// TIA Portal V15.1 export
// export: Created 2026-01-15T16:29:49.0596831Z, ExportSetting WithDefaults, WithReadOnly, DisplayName Totally Integrated Automation Portal, DisplayVersion V15.1 Update 8, DisplayName TIA Portal Openness, DisplayVersion V15.1 Update 8, DisplayName STEP 7 Professional, DisplayVersion V15.1 Update 8, DisplayName WinCC Advanced, DisplayVersion V15.1 Update 8
VAR_GLOBAL   // PLC tag table "Out_Put"
   "Q_CAN AP1" AT %Q4.0 : Bool;   // Output_Nồi trộn
   "Q_GAU COT LIEU" AT %Q0.5 : Bool;   // Output_Băng tải xiên
   Q_BTX AT %Q0.1 : Bool;   // Output_Băng tải ngang
   Q_BTN AT %Q0.2 : Bool;   // Output_Tang sấy cốt liệu
   "Q_TANG SAY" AT %Q0.3 : Bool;   // Output_Bơm dầu DO
   "Q_XA W_AG1" AT %Q4.2 : Bool;   // Output_Gàu tải cốt liệu nóng
   "Q_XA W_SB1" AT %Q4.5 : Bool;   // Output_Sàn rung cốt liệu
   "Q_BOM NUOC" AT %Q2.1 : Bool;   // Output_Gàu tải phụ F/D
   "Q_MO CUA" AT %Q2.2 : Bool;   // Output_Vít tải F/D
   "Q_XA CL5" AT %Q3.1 : Bool;   // Output_Bơm nạp hạt nhựa SBS
   "Q_DONG CUA" AT %Q2.3 : Bool;   // Output_Quạt gió lọc bụi
   Q_MNK AT %Q2.4 : Bool;   // Output_Bơm nước lọc bụi
   "Q_BOM SBS" AT %Q1.1 : Bool;   // Output_Van mở cửa nồi trộn
   "Q_CAN AG1" AT %Q3.2 : Bool;   // Output_Van đóng cửa nồi trộn
   "Q_VIT TAI FD" AT %Q1.0 : Bool;   // Output_Máy nén khí
   "Q_XA CL1" AT %Q2.5 : Bool;   // Output_Băng tải xả cốt liệu 1
   "Q_XA CL2" AT %Q2.6 : Bool;   // Output_Băng tải xả cốt liệu 2
   "Q_CAN AG2" AT %Q3.3 : Bool;   // Output_Băng tải xả cốt liệu 3
   "Q_XA CL3" AT %Q2.7 : Bool;   // Output_Băng tải xả cốt liệu 4
   "Q_XA CL4" AT %Q3.0 : Bool;   // Output_Băng tải xả cốt liệu 5
   "Q_CAN AG3" AT %Q3.4 : Bool;   // Output_Van cân AG1
   "Q_CAN AG4" AT %Q3.5 : Bool;   // Output_Van cân AG2
   "Q_CAN AG5" AT %Q3.6 : Bool;   // Output_Van cân AG3
   "Q_SAN RUNG" AT %Q0.6 : Bool;   // Output_Van cân AG4
   "Q_CAN FD1" AT %Q3.7 : Bool;   // Output_Van cân AG5
   "Q_CAN SB1" AT %Q4.1 : Bool;   // Output_Van cân F/D
   "Q_NOI TRON" AT %Q0.0 : Bool;   // Output_Bơm nhựa
   "Q_XA W_AP1" AT %Q4.4 : Bool;   // Output_Van cân hạt nhựa SBS
   "Q_XA W_FD1" AT %Q4.3 : Bool;   // Output_Van xả cân AG1
   "Q_BOM TUOI NHUA" AT %Q4.6 : Bool;   // Output_Van xả cân FD1
   "Q_DAU DOT" AT %Q4.7 : Bool;   // Output_Van xả cân AP1
   "Q_VAN XA SBS" AT %Q5.0 : Bool;   // Output_Van xả cân SB1
   "Q_Rung CL1" AT %Q5.1 : Bool;   // Output_Bổ ssung 1
   "Q_Rung CL2" AT %Q5.2 : Bool;   // Output_Bổ ssung 2
   "Q_Rung CL3" AT %Q5.3 : Bool;   // Output_Bổ ssung 3
   "Q_NOTE 7" AT %Q5.4 : Bool;   // Output_Bổ ssung 4
   "Q_QUAT GIO" AT %Q2.0 : Bool;   // Output_Bổ ssung 5
   "Q_GAU FD" AT %Q0.7 : Bool;   // Output_Bổ ssung 6
   "Q_BOM DAU" AT %Q0.4 : Bool;   // Output_Bổ ssung 7
   "NOI TRON" AT %M500.0 : Bool;   // Nồi trộn
   BTX AT %M500.1 : Bool;   // Băng tải xiên
   BTN AT %M500.2 : Bool;   // Băng tải ngang
   "TANG SAY" AT %M500.3 : Bool;   // Tang sấy cốt liệu
   "BOM DAU" AT %M500.4 : Bool;   // Bơm dầu DO
   "GAU COT LIEU" AT %M500.5 : Bool;   // Gàu tải cốt liệu nóng
   "SAN RUNG" AT %M500.6 : Bool;   // Sàn rung cốt liệu
   "GAU FD" AT %M500.7 : Bool;   // Gàu tải phụ F/D
   "VIT TAI FD" AT %M501.0 : Bool;   // Vít tải F/D
   "BOM SBS" AT %M501.1 : Bool;   // Bơm nạp hạt nhựa SBS
   "QUAT GIO" AT %M501.2 : Bool;   // Quạt gió lọc bụi
   "BOM NUOC" AT %M501.3 : Bool;   // Bơm nước lọc bụi
   "MO CUA" AT %M501.4 : Bool;   // Van mở cửa nồi trộn
   "DONG CUA" AT %M501.5 : Bool;   // Van đóng cửa nồi trộn
   MNK AT %M501.6 : Bool;   // Máy nén khí
   "XA CL1" AT %M501.7 : Bool;   // Băng tải xả cốt liệu 1
   "XA CL2" AT %M502.0 : Bool;   // Băng tải xả cốt liệu 2
   "XA CL3" AT %M502.1 : Bool;   // Băng tải xả cốt liệu 3
   "XA CL4" AT %M502.2 : Bool;   // Băng tải xả cốt liệu 4
   "XA CL5" AT %M502.3 : Bool;   // Băng tải xả cốt liệu 5
   "CAN AG1" AT %M502.4 : Bool;   // Van cân AG1
   "CAN AG2" AT %M502.5 : Bool;   // Van cân AG2
   "CAN AG3" AT %M502.6 : Bool;   // Van cân AG3
   "CAN AG4" AT %M502.7 : Bool;   // Van cân AG4
   "CAN AG5" AT %M503.0 : Bool;   // Van cân AG5
   "CAN FD1" AT %M503.1 : Bool;   // Van cân F/D
   "CAN AP1" AT %M503.2 : Bool;   // Bơm nhựa
   "CAN SB1" AT %M503.3 : Bool;   // Van cân hạt nhựa SBS
   "XA W_AG1" AT %M503.4 : Bool;   // Van xả cân AG1
   "XA W_FD1" AT %M503.5 : Bool;   // Van xả cân FD1
   "XA W_AP1" AT %M503.6 : Bool;   // Van xả cân AP1
   "XA W_SB1" AT %M503.7 : Bool;   // Van xả cân SB1
   "BOM TUOI NHUA" AT %M504.0 : Bool;   // Bổ ssung 1
   "DAU DOT" AT %M504.1 : Bool;   // Bổ ssung 2
   "VAN XA SBS" AT %M504.2 : Bool;   // Bổ ssung 3
   "RUNG CL1" AT %M504.3 : Bool;   // Bổ ssung 4
   "RUNG CL2" AT %M504.4 : Bool;   // Bổ ssung 5
   "RUNG CL3" AT %M504.5 : Bool;   // Bổ ssung 6
   "NOTE 7" AT %M504.6 : Bool;   // Bổ ssung 7
   "Q_XA W_IND AGG1" AT %Q6.0 : Bool;   // Mode=độc lập, Van xả cấn AGG1
   "Q_XA W_IND AGG2" AT %Q6.1 : Bool;   // Mode=độc lập, Van xả cấn AGG2
   "Q_XA W_IND AGG3" AT %Q6.2 : Bool;   // Mode=độc lập, Van xả cấn AGG3
   "Q_XA W_IND AGG4" AT %Q6.3 : Bool;   // Mode=độc lập, Van xả cấn AGG4
   "Q_XA W_IND AGG5" AT %Q6.4 : Bool;   // Mode=độc lập, Van xả cấn AGG5
END_VAR
